// TIA Portal V16 export
// export: Created 2022-02-04T14:40:23.6191179Z, ExportSetting WithDefaults, DisplayName Totally Integrated Automation Portal, DisplayVersion V16 Update 1, DisplayName TIA Portal Version Control Interface, DisplayVersion V16, DisplayName TIA Portal Openness, DisplayVersion V16, DisplayName SINAMICS Startdrive Advanced, DisplayVersion V16 Update 5, DisplayName SINAMICS Startdrive G130, G150, S120, S150, SINAMICS MV, S210, DisplayVersion V16 Update 5, DisplayName SINAMICS Startdrive G110M, G120, G120C, G120D, G120P, G115D, DisplayVersion V16 Update 5, DisplayName STEP 7 Professional, DisplayVersion V16, DisplayName STEP 7 Safety, DisplayVersion V16, DisplayName WinCC Advanced, DisplayVersion V16, DisplayName SIMATIC Visualization Architect, DisplayVersion V16
DATA_BLOCK "FB_Gasket_Carousel_DB"   // DB32
VERSION : 0.1
// stored: AutoNumber true, InstanceOfName FB_Gasket_Carousel, InstanceOfType FB
"FB_Gasket_Carousel"
   // VAR_INPUT
   //    make_layer : Bool;
   //    full_reset : Bool;
   //    pause : Bool;
   //    try_unpause : Bool;
   //    gasket_sensor : Bool;
   //    hook_sensor : Bool;
   //    last_hook_sensor : Bool;
   //    ramp_upper_sensor : Bool;
   //    gasket_cup_closed_sensor : Bool;
   //    no_ramp_flag : Bool;
   //    enable_double_schema : Bool;
   //    layer_num : Int;
   //    "2_schema_height" : Int;
   //    GASKET_PLACES_MAX : Int;
   //    HOOK_ENCODER_BARRIER : Int;
   //    GUARANTEED_HOOK_OFFSET : Int;
   //    OFFSET_DOWN_DEVICE : Int;
   //    OFFSET_LAST_HOOK : Int;
   //    OFFSET_LAYER_READY : Int;
   //    OFFSET_REVERS : Int;
   //    enc_pos : DInt;
   //    "1_schema_server" : DInt;
   //    "2_schema_server" : DInt;
   //    default_speed : Real;
   //    offset_speed : Real;
   //    default_reverse_speed : Real;
   // END_VAR
   // VAR_OUTPUT
   //    Carousel_FWD : Bool;
   //    Carousel_BWD : Bool;
   //    Ski_UP : Bool;
   //    Ski_DOWN : Bool;
   //    m_busy : Bool;
   //    m_acquire : Bool;
   //    m_released : Bool;
   //    ALM_NoGasketToUP : Bool;
   //    ALM_SensHook : Bool;
   //    ALM_SensLastHook : Bool;
   //    s_man_cntl : Bool;
   //    s_paused : Bool;
   //    Carousel_Speed : Real;
   // END_VAR
   // VAR RETAIN
   //    pos_defined : Bool;
   //    gasket_ready : Bool;
   //    _State : Int;
   //    s_max_hooks : Int;
   //    schema : DInt;
   //    enc_shot : DInt;
   //    hook_hold_timer : TOF;
   //    last_hook_hold_timer { S7_SetPoint := 'True'} : TOF;
   //    gasket_filter { S7_SetPoint := 'True'} : TON;
   //    Counters : Struct
   //       hooks : Int;
   //    END_STRUCT;
   //    Memento : Struct
   //       fwd : Bool;
   //       bwd : Bool;
   //       up : Bool;
   //       down : Bool;
   //       state : Int;
   //       speed : Real;
   //    END_STRUCT;
   //    SIG_old : Struct
   //       hook : Bool;
   //       last_hook : Bool;
   //    END_STRUCT;
   // END_VAR
BEGIN
END_DATA_BLOCK
